FUNCTION_BLOCK FB_SaMElementDiagnostics EXTENDS FB_SaMElement
VAR
END_VAR

END_FUNCTION_BLOCK

(* stored: Version 1.1.0.1
   POU FB_SaMElementDiagnostics: Id {ed2fdcb4-4966-0de9-308c-06dd2fbf700a}, SpecialFunc None *)
